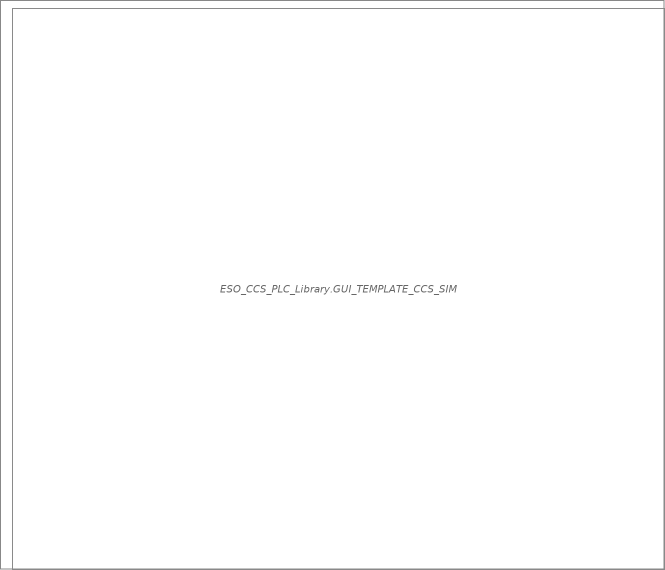
VISUALIZATION GUI_CCS_SIM  // 665x570
    Frame (12,8 653x562)
        shows ESO_CCS_PLC_Library.GUI_TEMPLATE_CCS_SIM(m_Instance := MAIN.ccs_sim)
END_VISUALIZATION

(* stored: Version 1.1.0.1, ProductVersion 3.1.4024.9
   Visu GUI_CCS_SIM: Id {fd9b18b7-02f2-4db4-b0e9-5c12c7c4f186} *)
